// TIA Portal V20 export
DATA_BLOCK "zGM SafetyGlobalChecksum_DB"   // DB5710
AUTHOR : TayNara
FAMILY : GM_CITI_3_2
VERSION : 1.0
// stored: InstanceOfName zGM SafetyGlobalChecksum, InstanceOfType FB
"zGM SafetyGlobalChecksum"
   // VAR_INPUT
   //    Start : Bool;
   //    ReadFrequency : Time;
   //    HardwareID_CU1 : HW_IO;
   //    HardwareID_CU2 : HW_IO;
   //    HardwareID_CU3 : HW_IO;
   //    HardwareID_CU4 : HW_IO;
   //    HardwareID_CU5 : HW_IO;
   //    HardwareID_CU6 : HW_IO;
   //    PlcSafetySignatureIn : DWord;
   // END_VAR
   // VAR_OUTPUT
   //    SingleSafetyChecksum : DWord;
   //    Busy : Bool;
   //    Error : Bool;
   // END_VAR
   // VAR
   //    instSinaParaS { S7_SetPoint := 'True'} : Array[1..6] of SinaParaS;
   //    statEnableReadSeq : Bool;
   //    statStartFN : Bool;
   //    statFreqTimer1 { S7_SetPoint := 'True'} : TON_TIME;
   //    statFreqTimer2 { S7_SetPoint := 'True'} : TON_TIME;
   //    statSafetyChecksum { S7_SetPoint := 'True'} : DWord;
   //    statTimeUp { S7_SetPoint := 'True'} : Bool;
   //    statTimeUpFP : Bool;
   //    statReadFrequency : Time;
   //    statResetEnableFP : Bool;
   // END_VAR
BEGIN
END_DATA_BLOCK
